// SIMATIC S7-200 project (STEP 7-Micro/WIN), CPU 221 REL 01.10

ORGANIZATION_BLOCK 主程序:OB1
TITLE=程序注释
BEGIN
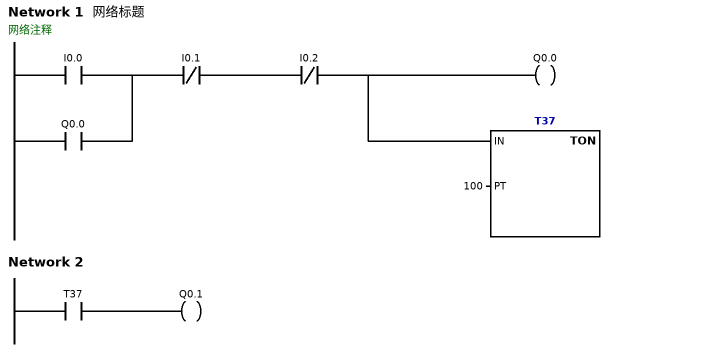
Network 1 // 网络标题
// 网络注释
// (network saved uncompiled; LAD cells follow)
// row 0: c0 -| |- I0.0 v  c1 -|/|- I0.1  c2 -|/|- I0.2 v  c3 --  c4 -( ) Q0.0
// row 1: c0 -| |- Q0.0 ^  c2 ^  c3 --  c4 [TON T37 IN:=power@row1, PT:=100]
// row 2: c4 [box]
Network 2
// (network saved uncompiled; LAD cells follow)
// row 0: c0 -| |- T37  c1 -( ) Q0.1
END_ORGANIZATION_BLOCK
